(* Logix 5000 project; controller Digital_Interlock_PLC vendor 1 type 14 code 196 rev 37.11; software revision 37.00; part 2 of 2 *)
(* tags used below, declared in another part *)
   Comms : UDT_Comms;
   CommsHealthy : BOOL;   // All machines are communicating
   PrefeederHBDetect : AOI_Detect_Heartbeat;
   PressHBDetect : AOI_Detect_Heartbeat;
   StackerHBDetect : AOI_Detect_Heartbeat;
   _DEBUG : BOOL;
   CommsStatus : DINT;
   EnableLineOptimization : BOOL;
   FromPrefeeder : DINT[33];   // DINTs used: 0-2
   FromPress : DINT[33];
   FromStacker : DINT[33];   // DINTS used: 0-22
   PrefeederData : UDT_MSG;
   PrefeederLFO : UDT_MachineLFOProperties;
   PrefeederLFO_AOI : AOI_Optimize_Flow;
   PressLFO : UDT_MachineLFOProperties;
   PressLFO_AOI : AOI_Optimize_Flow;
   StackerLFO : UDT_MachineLFOProperties;
   StackerLFO_AOI : AOI_Optimize_Flow;
(* MainProgram, continued *)

   //PR1:O.Data[22] := FromStacker[16]; 			//(Stacker -> Press) fromStacker.PrintStation[1].fltDesiredSidewaysAdjust REAL
   //PR1:O.Data[23] := FromStacker[17]; 			//(Stacker -> Press) fromStacker.PrintStation[2].fltDesiredSidewaysAdjust REAL
   //PR1:O.Data[24] := FromStacker[18]; 			//(Stacker -> Press) fromStacker.PrintStation[3].fltDesiredSidewaysAdjust REAL
   //PR1:O.Data[25] := FromStacker[19]; 			//(Stacker -> Press) fromStacker.PrintStation[4].fltDesiredSidewaysAdjust REAL
   //PR1:O.Data[26] := FromStacker[20]; 			//(Stacker -> Press) fromStacker.PrintStation[5].fltDesiredSidewaysAdjust REAL
   //PR1:O.Data[27] := FromStacker[21]; 			//(Stacker -> Press) fromStacker.PrintStation[6].fltDesiredSidewaysAdjust REAL
   //PR1:O.Data[28] := FromStacker[22]; 			//(Stacker -> Press) fromStacker.PrintStation[7].fltDesiredSidewaysAdjust REAL
   #endregion
   
   #region CURRENT SPEEDS
   //PrefeederLFO.CurrentSpeed := FromPrefeeder[1]; 				//(Pre-Feeder -> Interlock) FromPrefeeder.CurrentSpeed INT
   //PressLFO.CurrentSpeed := PR1:I.Data[2];						//(Press -> Interlock) FromPress.CurrentSpeed
   //StackerLFO.CurrentSpeed := ST1:I.Data[1]; 					//(Stacker -> Interlock) fromStacker.CurrentSpeed INT
   #endregion
   
   #region PATTERN MAX SPEEDS
   //PrefeederLFO.PatternMaxSpeed := FromPrefeeder[2]; 			//(Pre-Feeder -> Interlock) FromPrefeeder.PatternMaxSpeed INT
   //PressLFO.PatternMaxSpeed := FromPress[23];					//(Press -> Interlock) FromPress.PatternMaxSpeed INT
   //StackerLFO.PatternMaxSpeed := ST1:I.Data[2]; 				//(Stacker -> Interlock) fromStacker.PatternMaxSpeed INT
   #endregion
END_ROUTINE

ROUTINE MonitorCommsRoutine   (* ladder *)
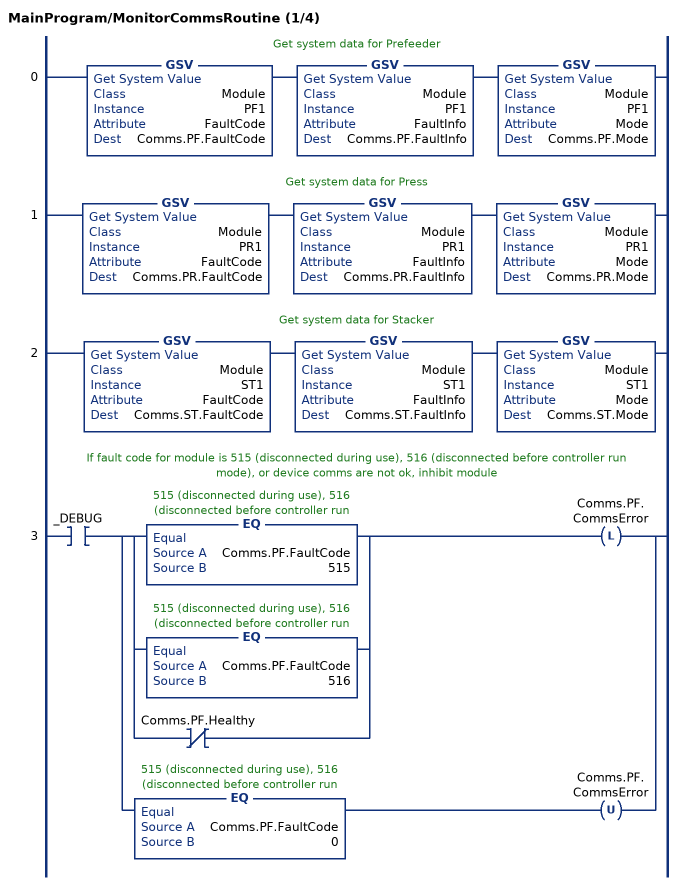
   // Get system data for Prefeeder
   0: GSV(Module,PF1,FaultCode,Comms.PF.FaultCode)GSV(Module,PF1,FaultInfo,Comms.PF.FaultInfo)GSV(Module,PF1,Mode,Comms.PF.Mode);
   // Get system data for Press
   1: GSV(Module,PR1,FaultCode,Comms.PR.FaultCode)GSV(Module,PR1,FaultInfo,Comms.PR.FaultInfo)GSV(Module,PR1,Mode,Comms.PR.Mode);
   // Get system data for Stacker
   2: GSV(Module,ST1,FaultCode,Comms.ST.FaultCode)GSV(Module,ST1,FaultInfo,Comms.ST.FaultInfo)GSV(Module,ST1,Mode,Comms.ST.Mode);
   // If fault code for module is 515 (disconnected during use), 516 (disconnected before controller run mode), or device comms are not ok, inhibit module
   3: XIC(_DEBUG)[[EQ(Comms.PF.FaultCode,515) ,EQ(Comms.PF.FaultCode,516) ,XIO(Comms.PF.Healthy) ] OTL(Comms.PF.CommsError) ,EQ(Comms.PF.FaultCode,0) OTU(Comms.PF.CommsError) ];
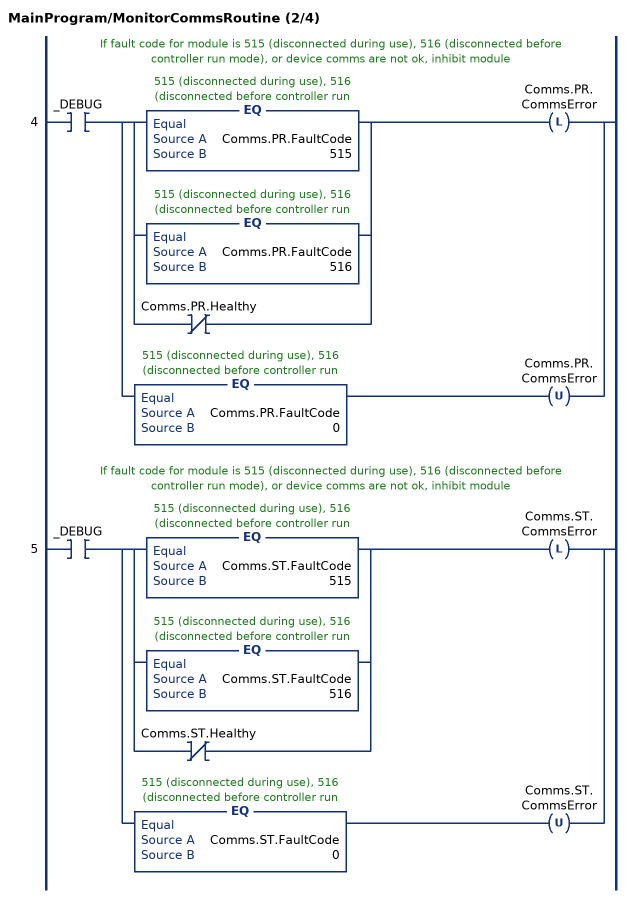
   // If fault code for module is 515 (disconnected during use), 516 (disconnected before controller run mode), or device comms are not ok, inhibit module
   4: XIC(_DEBUG)[[EQ(Comms.PR.FaultCode,515) ,EQ(Comms.PR.FaultCode,516) ,XIO(Comms.PR.Healthy) ] OTL(Comms.PR.CommsError) ,EQ(Comms.PR.FaultCode,0) OTU(Comms.PR.CommsError) ];
   // If fault code for module is 515 (disconnected during use), 516 (disconnected before controller run mode), or device comms are not ok, inhibit module
   5: XIC(_DEBUG)[[EQ(Comms.ST.FaultCode,515) ,EQ(Comms.ST.FaultCode,516) ,XIO(Comms.ST.Healthy) ] OTL(Comms.ST.CommsError) ,EQ(Comms.ST.FaultCode,0) OTU(Comms.ST.CommsError) ];
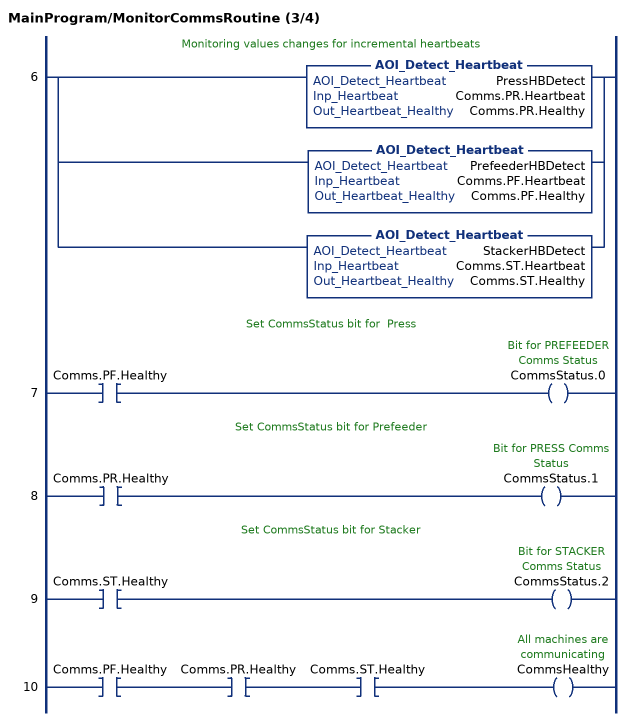
   // Monitoring values changes for incremental heartbeats
   6: [AOI_Detect_Heartbeat(PressHBDetect,Comms.PR.Heartbeat,Comms.PR.Healthy) ,AOI_Detect_Heartbeat(PrefeederHBDetect,Comms.PF.Heartbeat,Comms.PF.Healthy) ,AOI_Detect_Heartbeat(StackerHBDetect,Comms.ST.Heartbeat,Comms.ST.Healthy) ];
   // Set CommsStatus bit for  Press
   7: XIC(Comms.PF.Healthy)OTE(CommsStatus.0);
   // Set CommsStatus bit for Prefeeder
   8: XIC(Comms.PR.Healthy)OTE(CommsStatus.1);
   // Set CommsStatus bit for Stacker
   9: XIC(Comms.ST.Healthy)OTE(CommsStatus.2);
   10: XIC(Comms.PF.Healthy)XIC(Comms.PR.Healthy)XIC(Comms.ST.Healthy)OTE(CommsHealthy);
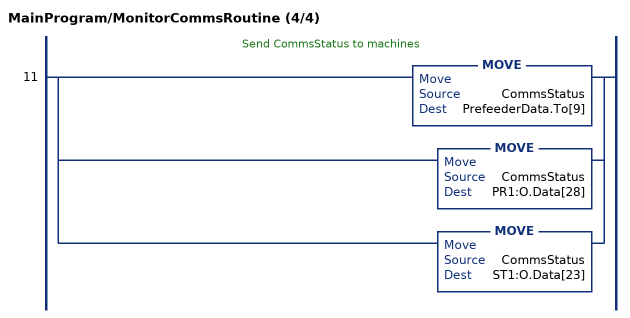
   // Send CommsStatus to machines
   11: [MOVE(CommsStatus,PrefeederData.To[9]) ,MOVE(CommsStatus,PR1:O.Data[28]) ,MOVE(CommsStatus,ST1:O.Data[23]) ];
END_ROUTINE
END_PROGRAM

PROGRAM ManageOptimizationProgram   (* main routine MainRoutine *)
// Program containing routines for Line Flow Optimization.

ROUTINE MainRoutine   (* ladder *)
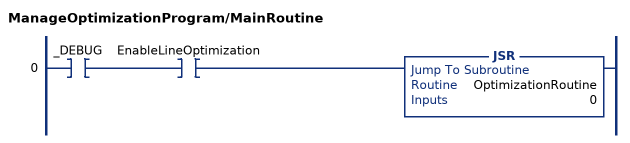
   0: XIC(_DEBUG)XIC(EnableLineOptimization)JSR(OptimizationRoutine,0);
END_ROUTINE

ROUTINE OptimizationRoutine   (* ladder *)
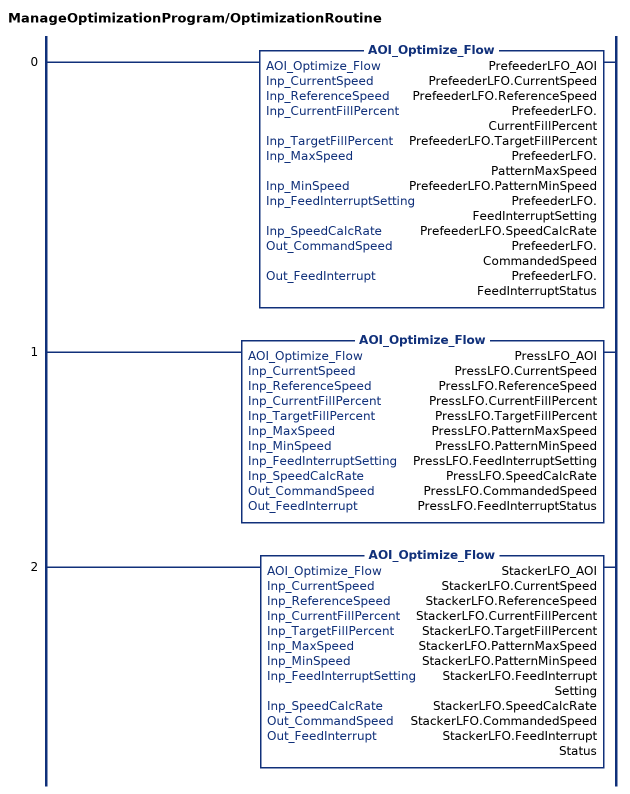
   0: AOI_Optimize_Flow(PrefeederLFO_AOI,PrefeederLFO.CurrentSpeed,PrefeederLFO.ReferenceSpeed,PrefeederLFO.CurrentFillPercent,PrefeederLFO.TargetFillPercent,PrefeederLFO.PatternMaxSpeed,PrefeederLFO.PatternMinSpeed,PrefeederLFO.FeedInterruptSetting,PrefeederLFO.SpeedCalcRate,PrefeederLFO.CommandedSpeed,PrefeederLFO.FeedInterruptStatus);
   1: AOI_Optimize_Flow(PressLFO_AOI,PressLFO.CurrentSpeed,PressLFO.ReferenceSpeed,PressLFO.CurrentFillPercent,PressLFO.TargetFillPercent,PressLFO.PatternMaxSpeed,PressLFO.PatternMinSpeed,PressLFO.FeedInterruptSetting,PressLFO.SpeedCalcRate,PressLFO.CommandedSpeed,PressLFO.FeedInterruptStatus);
   2: AOI_Optimize_Flow(StackerLFO_AOI,StackerLFO.CurrentSpeed,StackerLFO.ReferenceSpeed,StackerLFO.CurrentFillPercent,StackerLFO.TargetFillPercent,StackerLFO.PatternMaxSpeed,StackerLFO.PatternMinSpeed,StackerLFO.FeedInterruptSetting,StackerLFO.SpeedCalcRate,StackerLFO.CommandedSpeed,StackerLFO.FeedInterruptStatus);
END_ROUTINE
END_PROGRAM
